// TwinCAT 3 PLC project ServerSampleProject
// ProgramVersion: 3.1.4026.13
// libraries:
//   Tc2_Standard, * (Beckhoff Automation GmbH)
//   Tc2_System, * (Beckhoff Automation GmbH)
//   Tc3_Module, * (Beckhoff Automation GmbH)
// project tree:
//   DUTs/ ST_Structure.TcDUT, ST_SubStructure.TcDUT
//   / PlcTask.TcTTO
//   POUs/ FB_Mathematics.TcPOU, MAIN.TcPOU
// real-time tasks:
//   TASK PlcTask: cycle T#10ms, priority 20, ADS port 350

CONFIGURATION ServerSampleProject
    RESOURCE PLC ON TwinCAT3
        TASK PlcTask(INTERVAL := T#10ms, PRIORITY := 20);
        PROGRAM MAIN WITH PlcTask : MAIN;
    END_RESOURCE
END_CONFIGURATION

// ---- DUTs/ST_Structure.TcDUT
TYPE ST_Structure :
STRUCT
	a : INT;
	b : DINT;
	c : ARRAY[0..9] OF REAL;
	{attribute 'OPC.UA.DA.StructuredType':='1'}
	d : ST_SubStructure;
END_STRUCT
END_TYPE

// ---- DUTs/ST_SubStructure.TcDUT
TYPE ST_SubStructure :
STRUCT
	e : LREAL;
	f : DT;
END_STRUCT
END_TYPE

// ---- POUs/MAIN.TcPOU
PROGRAM MAIN
VAR
	{attribute 'OPC.UA.DA':='1'}
	nCounter : INT;
	
	{attribute 'OPC.UA.DA':='1'}
	nNumber : INT;
	
	{attribute 'OPC.UA.DA':='1'}
	fbMathematics : FB_Mathematics;
	
	{attribute 'OPC.UA.DA':='1'}
	iVar1 : INT := 42;
	
	{attribute 'OPC.UA.DA':='1'}
	iVar2 : INT := 43;
	
	{attribute 'OPC.UA.DA':='1'}
	{attribute 'OPC.UA.DA.Access':='1'}
	iVar3_readOnly : INT := 43;	
	
	{attribute 'OPC.UA.DA':='1'}
	{attribute 'OPC.UA.DA.Description' := 'Some description'} 
	iArrayIntVar1 : ARRAY[0..9] OF INT := [10(42)];
	
	{attribute 'OPC.UA.DA':='1'}
	iArrayIntVar2 : ARRAY[0..11] OF INT := [12(41)];	
	
	{attribute 'OPC.UA.DA':='1'}
	iArrayIntVar3 : ARRAY[0..9] OF DINT;
	
	{attribute 'OPC.UA.DA':='1'}
	{attribute 'OPC.UA.DA.StructuredType':='1'}
	stStructure : ST_Structure;
	
	// Variable for HistoryUpdate (single) client sample
	{attribute 'OPC.UA.DA' := '1'}
	nMyValue : INT;
	
	// Variable for HistoryUpdate (multiple) client sample
	{attribute 'OPC.UA.DA' := '1'}
	nMyValue1 : INT;	
	{attribute 'OPC.UA.DA' := '1'}
	nMyValue2 : INT;
	{attribute 'OPC.UA.DA' := '1'}
	fMyValue3 : LREAL;	
END_VAR

nCounter := nCounter + 1;

END_PROGRAM

// ---- POUs/FB_Mathematics.TcPOU
FUNCTION_BLOCK FB_Mathematics
VAR_INPUT
END_VAR
VAR_OUTPUT
END_VAR
VAR
	{attribute 'OPC.UA.DA':='1'}
	nNumberOfCallsMMul : INT;
	
	{attribute 'OPC.UA.DA':='1'}
	nNumberOfCallsMNoArgs : INT;
END_VAR

{attribute 'TcRpcEnable':='1'}
METHOD M_Mul : DINT
VAR_INPUT
	a : INT;
	b : INT;
END_VAR
M_Mul := a * b;
nNumberOfCallsMMul := nNumberOfCallsMMul + 1;
END_METHOD

{attribute 'TcRpcEnable':='1'}
METHOD M_NoArgs
VAR_INPUT
END_VAR
nNumberOfCallsMNoArgs := nNumberOfCallsMNoArgs + 1;
END_METHOD

END_FUNCTION_BLOCK
